// TIA Portal V20 export
DATA_BLOCK "ControlNodes"   // DB143
// stored: MemoryReserve 100, Namespace Unit1.Em0
   VAR
      em : "LAF_typeEmControlNode";
      emstate { S7_SetPoint := 'True'} : "LUC_typeStates";
      cm : "Unit1.Em0.typeCmControlNode";
      citiMap : Struct
         PMC : "LER_PMC_Input_Data";
         FlexNet { S7_SetPoint := 'True'} : "LER_FlexNet_Data";
      END_STRUCT;
      stacker1NgBox : "Unit1.Em0.typeSequenceControlNode";
      SpecialFunctionMode : Struct
         DryRun : Struct
            JRdetectPV : Array[0..15] of Bool;
         END_STRUCT;
      END_STRUCT;
      unitCommunication : "Unit1.Em0.typeUnitCommunicationControlNode";
      cmStacker1NgBoxDetect : "LBC_typeDigitalSignalControlNode";
      cmStacker1NgBoxFullDetect : "LBC_typeDigitalSignalControlNode";
      cmStacker1NgBoxLoadingUpDown : "LBC_typeTwoWayActuatorControlNode";
      cmStacker1NgBoxUnitMoverBwdFwd : "LBC_typeTwoWayActuatorControlNode";
      cmStacker1NgBoxClampLeftOpenClose : "LBC_typeTwoWayActuatorControlNode";
      cmStacker1NgBoxClampRightOpenClose : "LBC_typeTwoWayActuatorControlNode";
      cmStacker1NgBoxClampMoverOpenClose : "LBC_typeTwoWayActuatorControlNode";
      cmStacker1NgBoxLiftDownUp : "LBC_typeTwoWayActuatorControlNode";
      cmStacker1NgBoxLockDownUp : "LBC_typeTwoWayActuatorControlNode";
   END_VAR
BEGIN
   // cmStacker1NgBoxLoadingUpDown.commands.commandHomePos : STAKC #1 NG CLAMP Z-AXIS UP
   // cmStacker1NgBoxLoadingUpDown.commands.commandWorkPos : STAKC #1 NG CLAMP Z-AXIS DOWN
   // cmStacker1NgBoxUnitMoverBwdFwd.commands.commandHomePos : STAKC #1 NG CLAMP UNIT MOVER BACKWARD
   // cmStacker1NgBoxUnitMoverBwdFwd.commands.commandWorkPos : STAKC #1 NG CLAMP UNIT MOVER FORWARD
   // cmStacker1NgBoxClampLeftOpenClose.commands.commandHomePos : STACK #1 NG CLAMP LEFT OPEN
   // cmStacker1NgBoxClampLeftOpenClose.commands.commandWorkPos : STACK #1 NG CLAMP LEFT CLOSE
   // cmStacker1NgBoxClampRightOpenClose.commands.commandHomePos : STACK #1 NG CLAMP RIGHT OPEN
   // cmStacker1NgBoxClampRightOpenClose.commands.commandWorkPos : STACK #1 NG CLAMP RIGHT CLOSE
   // cmStacker1NgBoxLiftDownUp.commands.commandHomePos : STACK #1 NG BOX LIFT UP
   // cmStacker1NgBoxLiftDownUp.commands.commandWorkPos : STACK #1 NG BOX LIFT DOWN
   // cmStacker1NgBoxLockDownUp.commands.commandHomePos : STACK #1 NG BOX LOCK DOWN
   // cmStacker1NgBoxLockDownUp.commands.commandWorkPos : STACK #1 NG BOX LOCK UP
END_DATA_BLOCK
